Universal Robots PolyScope program: Move_Circle.urp

Program Move_Circle (installation=default directory=/home/ur/ursim-current/programs/new folder_1 createdIn=5.11.4.108353 lastSavedIn=5.11.4.108353 robotSerialNumber=20195299999)
Calibrated DH parameters: a=[0, -0.6127, -0.57155, 0, 0, 0]; d=[0.1807, 0, 0, 0.17415, 0.11985, 0.11655]; alpha=[1.570796, 0, 0, 1.570796, -1.570796, 0]; deltaTheta=[0, 0, 0, 0, 0, 0]
BeforeStart
  MoveJ speed 60 deg/s, acceleration 80 deg/s^2 (useActiveTCP=true) feature=Base
    Waypoint Waypoint_Home: TCP in base x=0.027 y=-700.008 z=307.642 mm, rx=0.0687 ry=3.1392 rz=0.0004 rad; joints [-75.608, -100.646, -118.225, -51.12, 90.093, 16.898] deg
  v_radius := 0.050
  v_point_1 := p[Waypoint_Home[0] + v_radius,Waypoint_Home[1],Waypoint_Home[2],Waypoint_Home[3],Waypoint_Home[4],Waypoint_Home[5]]
  v_point_2 := p[Waypoint_Home[0],Waypoint_Home[1] + v_radius,Waypoint_Home[2],Waypoint_Home[3],Waypoint_Home[4],Waypoint_Home[5]]
  v_point_3 := p[Waypoint_Home[0] - v_radius,Waypoint_Home[1],Waypoint_Home[2],Waypoint_Home[3],Waypoint_Home[4],Waypoint_Home[5]]
  v_point_4 := p[Waypoint_Home[0],Waypoint_Home[1] - v_radius,Waypoint_Home[2],Waypoint_Home[3],Waypoint_Home[4],Waypoint_Home[5]]
Robot Program (runOnlyOnce=false)
  MoveP speed 250 mm/s, acceleration 1200 mm/s^2 (blendRadius=0.025 useActiveTCP=true) feature=Base
    Waypoint Waypoint (Variable): variable=v_point_1
    CircleMove (OrientationMode=UNCONSTRAINED)
      Waypoint Waypoint (Variable): variable=v_point_2
      Waypoint Waypoint (Variable): variable=v_point_3
    CircleMove (OrientationMode=UNCONSTRAINED)
      Waypoint Waypoint (Variable): variable=v_point_4
      Waypoint Waypoint (Variable): variable=v_point_1
